// TIA Portal V19 export
TYPE "Prod_Beam_Area"
   STRUCT
      Halted { ExternalWritable := 'False'} : "Prod_Halted";
      Man { ExternalWritable := 'False'} : Bool;
      Doors_Closed { ExternalWritable := 'False'} : Bool;
      CycleON { ExternalWritable := 'False'} : Bool;
      Running { ExternalWritable := 'False'} : Bool;
      SetUpDone : Bool;
      SetupDone_Ax : Array[1..9] of Bool;
   END_STRUCT;
END_TYPE
